ABB RobotStudio station: Mark 4.rspag

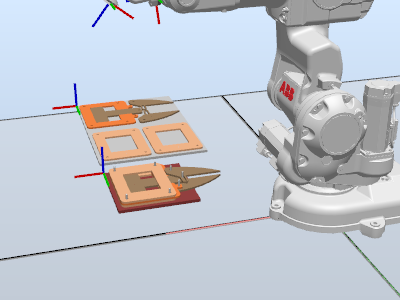
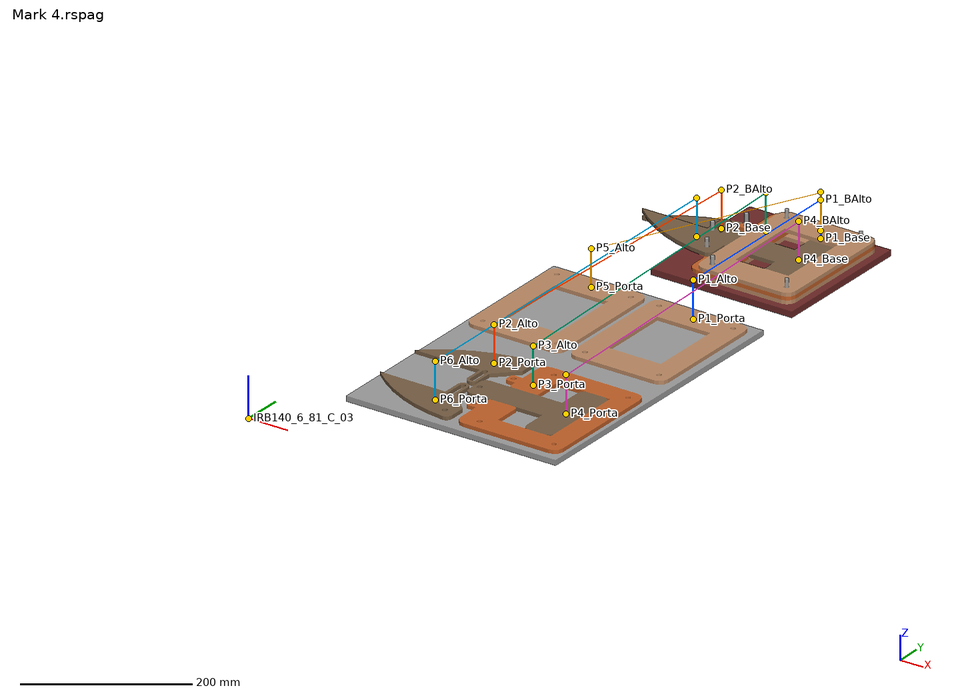
[picture v1: parts stored in the station drawn from their meshes, with robot base, taught points and paths (robot models come from the ABB library and are not in the file)]
--- station ---
Station Mark 4 (saved by RobotStudio 22.2.9947.0)
Controller Mark4_PF
  mechanical unit ROB_1: IRB140_6_81_C_03, 6 joints, base frame (0, 0, 0) mm
Layout (positions relative to the parent item):
  - IRB140_6_81_C_03 [mechanism, from Robots\IRB140_6_81_C_G_03.rslib] at (0, 0, 0) mm; joint values [0, 0, 0, 0, 0.1225, 0] (rad or m)
  - Base [part] at (585, 215, 277) mm, rotated rx 0 ry 0 rz 180 deg, size 282.5 x 200 x 35 mm
  - Portapiezas [part] at (550, -150, 277) mm, rotated rx 0 ry 0 rz 180 deg, size 297 x 420 x 12 mm
  - Tool_AJDJ [mechanism] at (514.51, 0, 704.06) mm, rotated rx 180 ry 82.98 rz 180 deg
      TCP Tool_AJDJ at (-6, 0, 116) mm, rotated rx 0 ry 45 rz 0 deg
      links: Herramienta
Attachment: Tool_AJDJ is attached to IRB140_6_81_C_03 / Link6

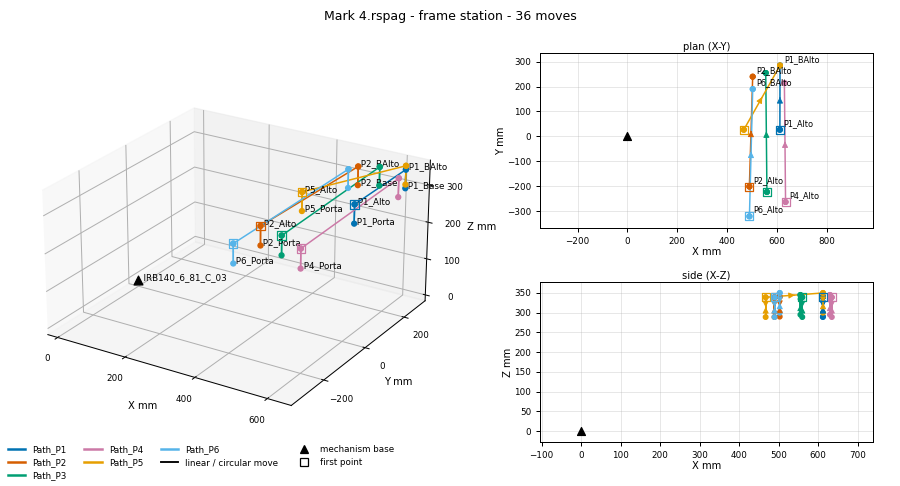
[picture p0: tool path of Mark 4.rspag in frame station, 36 of 39 moves have a stored position in this frame; points joined in program order, loops and branches not executed]
--- Backups/Mark4_PF/RAPID/TASK1/PROGMOD/CalibData.mod ---
MODULE CalibData
    PERS tooldata Tool_AJDJ:=[TRUE,[[-6,0,116],[0.923879533,0,0.382683432,0]],[0.15,[0,0,1],[1,0,0,0],0,0,0]];
    TASK PERS wobjdata Portapiezas:=[FALSE,TRUE,"",[[688.989,-362.504,284],[1,0,0,0]],[[0,0,0],[1,0,0,0]]];
    TASK PERS wobjdata BaseG:=[FALSE,TRUE,"",[[689.264,115.06,285],[1,0,0,0]],[[0,0,0],[1,0,0,0]]];
ENDMODULE

--- Backups/Mark4_PF/RAPID/TASK1/PROGMOD/Module1.mod ---
MODULE Module1
    CONST jointtarget HomeHerramienta:=[[0,0,0,0,45,0],[9E+09,9E+09,9E+09,9E+09,9E+09,9E+09]];
    CONST robtarget P1_Alto:=[[-77.3,389.019,55],[0,0,1,0],[0,-1,0,0],[9E+09,9E+09,9E+09,9E+09,9E+09,9E+09]];
    CONST robtarget P1_Porta:=[[-77.3,389.019,5],[0,0,1,0],[0,-2,1,0],[9E+09,9E+09,9E+09,9E+09,9E+09,9E+09]];
    CONST robtarget P1_BAlto:=[[-77.1,169.1,55],[0,0,1,0],[0,-1,0,0],[9E+09,9E+09,9E+09,9E+09,9E+09,9E+09]];
    CONST robtarget P1_Base:=[[-77.1,169.1,5],[0,0,1,0],[0,-1,0,0],[9E+09,9E+09,9E+09,9E+09,9E+09,9E+09]];
    CONST jointtarget HomeLaboratorio:=[[0,0,0,0,0,0],[9E+09,9E+09,9E+09,9E+09,9E+09,9E+09]];
    CONST robtarget P2_Alto:=[[-199.7,161,55],[0,0,1,0],[-1,0,-1,0],[9E+09,9E+09,9E+09,9E+09,9E+09,9E+09]];
    CONST robtarget P2_Porta:=[[-199.7,161,5],[0,0,1,0],[-1,1,-2,0],[9E+09,9E+09,9E+09,9E+09,9E+09,9E+09]];
    CONST robtarget P2_BAlto:=[[-186.7,124.4,55],[0,0,1,0],[0,-1,0,0],[9E+09,9E+09,9E+09,9E+09,9E+09,9E+09]];
    CONST robtarget P2_Base:=[[-186.7,124.4,5],[0,0,1,0],[0,-1,1,0],[9E+09,9E+09,9E+09,9E+09,9E+09,9E+09]];
    CONST robtarget P3_Alto:=[[-129.3,139.3,55],[0,0,1,0],[-1,0,-1,0],[9E+09,9E+09,9E+09,9E+09,9E+09,9E+09]];
    CONST robtarget P3_Porta:=[[-129.3,139.3,5],[0,0,1,0],[-1,0,-2,0],[9E+09,9E+09,9E+09,9E+09,9E+09,9E+09]];
    CONST robtarget P3_BAlto:=[[-134.3,139.3,60],[0,0,1,0],[0,-1,0,0],[9E+09,9E+09,9E+09,9E+09,9E+09,9E+09]];
    CONST robtarget P3_Base:=[[-134.3,139.3,10],[0,0,1,0],[0,-1,1,0],[9E+09,9E+09,9E+09,9E+09,9E+09,9E+09]];
    CONST robtarget P4_Alto:=[[-54.5,99.1,55],[0,0,1,0],[-1,0,-1,0],[9E+09,9E+09,9E+09,9E+09,9E+09,9E+09]];
    CONST robtarget P4_Porta:=[[-54.5,99.1,5],[0,0,1,0],[-1,0,-1,0],[9E+09,9E+09,9E+09,9E+09,9E+09,9E+09]];
    CONST robtarget P4_BAlto:=[[-59.5,99.1,60],[0,0,1,0],[0,-1,0,0],[9E+09,9E+09,9E+09,9E+09,9E+09,9E+09]];
    CONST robtarget P4_Base:=[[-59.5,99.1,10],[0,0,1,0],[0,-1,0,0],[9E+09,9E+09,9E+09,9E+09,9E+09,9E+09]];
    CONST robtarget P5_Alto:=[[-222,389.1,55],[0,0,1,0],[0,-1,0,0],[9E+09,9E+09,9E+09,9E+09,9E+09,9E+09]];
    CONST robtarget P5_Porta:=[[-222,389.1,5],[0,0,1,0],[0,-2,1,0],[9E+09,9E+09,9E+09,9E+09,9E+09,9E+09]];
    CONST robtarget P5_BAlto:=[[-77.1,169.1,65],[0,0,1,0],[0,-1,0,0],[9E+09,9E+09,9E+09,9E+09,9E+09,9E+09]];
    CONST robtarget P5_Base:=[[-77.1,169.1,15],[0,0,1,0],[0,-1,0,0],[9E+09,9E+09,9E+09,9E+09,9E+09,9E+09]];
    CONST robtarget P6_Alto:=[[-199.5,41.5,55],[0,0,1,0],[-1,0,-2,0],[9E+09,9E+09,9E+09,9E+09,9E+09,9E+09]];
    CONST robtarget P6_Porta:=[[-199.5,41.5,5],[0,0,1,0],[-1,0,-2,0],[9E+09,9E+09,9E+09,9E+09,9E+09,9E+09]];
    CONST robtarget P6_BAlto:=[[-186.6,74.6,65],[0,0,1,0],[0,-1,0,0],[9E+09,9E+09,9E+09,9E+09,9E+09,9E+09]];
    CONST robtarget P6_Base:=[[-186.6,74.6,15],[0,0,1,0],[0,-1,1,0],[9E+09,9E+09,9E+09,9E+09,9E+09,9E+09]];
    PROC ToHome()
        MoveAbsJ HomeLaboratorio,v150,z10,Tool_AJDJ\WObj:=BaseG;
    ENDPROC
    PROC Path_P1()
        MoveAbsJ HomeHerramienta,v150,z10,Tool_AJDJ\WObj:=BaseG;
        MoveL P1_Alto,v150,z10,Tool_AJDJ\WObj:=Portapiezas;
        MoveL P1_Porta,v50,z10,Tool_AJDJ\WObj:=Portapiezas;
        WaitDI DI_01,1;
        SetDO DO_01,1;
        WaitTime 0.05;
        SetDO DO_01,0;
        MoveL P1_Alto,v50,z10,Tool_AJDJ\WObj:=Portapiezas;
        MoveL P1_BAlto,v150,z10,Tool_AJDJ\WObj:=BaseG;
        MoveL P1_Base,v50,z10,Tool_AJDJ\WObj:=BaseG;
        WaitDI DI_01,1;
        SetDO DO_02,1;
        WaitTime 0.05;
        SetDO DO_02,0;
        MoveL P1_BAlto,v50,z10,Tool_AJDJ\WObj:=BaseG;
    ENDPROC
    PROC Path_P2()
        MoveL P2_Alto,v150,z10,Tool_AJDJ\WObj:=Portapiezas;
        MoveL P2_Porta,v50,z10,Tool_AJDJ\WObj:=Portapiezas;
        WaitDI DI_01,1;
        SetDO DO_01,1;
        WaitTime 0.05;
        SetDO DO_01,0;
        MoveL P2_Alto,v50,z10,Tool_AJDJ\WObj:=Portapiezas;
        MoveL P2_BAlto,v150,z10,Tool_AJDJ\WObj:=BaseG;
        MoveL P2_Base,v50,z10,Tool_AJDJ\WObj:=BaseG;
        WaitDI DI_01,1;
        SetDO DO_02,1;
        WaitTime 0.05;
        SetDO DO_02,0;
        MoveL P2_BAlto,v50,z10,Tool_AJDJ\WObj:=BaseG;
    ENDPROC
    PROC Path_P3()
        MoveL P3_Alto,v150,z10,Tool_AJDJ\WObj:=Portapiezas;
        MoveL P3_Porta,v50,z10,Tool_AJDJ\WObj:=Portapiezas;
        WaitDI DI_01,1;
        SetDO DO_01,1;
        WaitTime 0.05;
        SetDO DO_01,0;
        MoveL P3_Alto,v50,z10,Tool_AJDJ\WObj:=Portapiezas;
        MoveL P3_BAlto,v150,z10,Tool_AJDJ\WObj:=BaseG;
        MoveL P3_Base,v50,z10,Tool_AJDJ\WObj:=BaseG;
        WaitDI DI_01,1;
        SetDO DO_02,1;
        WaitTime 0.05;
        SetDO DO_02,0;
        MoveL P3_BAlto,v50,z10,Tool_AJDJ\WObj:=BaseG;
    ENDPROC
    PROC Path_P4()
        MoveL P4_Alto,v150,z10,Tool_AJDJ\WObj:=Portapiezas;
        MoveL P4_Porta,v50,z10,Tool_AJDJ\WObj:=Portapiezas;
        WaitDI DI_01,1;
        SetDO DO_01,1;
        WaitTime 0.05;
        SetDO DO_01,0;
        MoveL P4_Alto,v50,z10,Tool_AJDJ\WObj:=Portapiezas;
        MoveL P4_BAlto,v150,z10,Tool_AJDJ\WObj:=BaseG;
        MoveL P4_Base,v50,z10,Tool_AJDJ\WObj:=BaseG;
        WaitDI DI_01,1;
        SetDO DO_02,1;
        WaitTime 0.05;
        SetDO DO_02,0;
        MoveL P4_BAlto,v50,z10,Tool_AJDJ\WObj:=BaseG;
    ENDPROC
    PROC Path_P5()
        MoveL P5_Alto,v150,z10,Tool_AJDJ\WObj:=Portapiezas;
        MoveL P5_Porta,v50,z10,Tool_AJDJ\WObj:=Portapiezas;
        WaitDI DI_01,1;
        SetDO DO_01,1;
        WaitTime 0.05;
        SetDO DO_01,0;
        MoveL P5_Alto,v50,z10,Tool_AJDJ\WObj:=Portapiezas;
        MoveL P5_BAlto,v150,z10,Tool_AJDJ\WObj:=BaseG;
        MoveL P5_Base,v50,z10,Tool_AJDJ\WObj:=BaseG;
        WaitDI DI_01,1;
        SetDO DO_02,1;
        WaitTime 0.05;
        SetDO DO_02,0;
        MoveL P5_BAlto,v50,z10,Tool_AJDJ\WObj:=BaseG;
    ENDPROC
    PROC Path_P6()
        MoveL P6_Alto,v150,z10,Tool_AJDJ\WObj:=Portapiezas;
        MoveL P6_Porta,v50,z10,Tool_AJDJ\WObj:=Portapiezas;
        WaitDI DI_01,1;
        SetDO DO_01,1;
        WaitTime 0.05;
        SetDO DO_01,0;
        MoveL P6_Alto,v50,z10,Tool_AJDJ\WObj:=Portapiezas;
        MoveL P6_BAlto,v150,z10,Tool_AJDJ\WObj:=BaseG;
        MoveL P6_Base,v50,z10,Tool_AJDJ\WObj:=BaseG;
        WaitDI DI_01,1;
        SetDO DO_02,1;
        WaitTime 0.05;
        SetDO DO_02,0;
        MoveL P6_BAlto,v50,z10,Tool_AJDJ\WObj:=BaseG;
        MoveAbsJ HomeHerramienta,v150,z10,Tool_AJDJ\WObj:=BaseG;
    ENDPROC
    PROC main()
        SpyStart "HOME:/spy.log";
        SetDO DO_03,0;
        WaitDI DI_01,1;
        ToHome;
        WaitDI DI_01,1;
        Path_P1;
        Path_P2;
        Path_P3;
        Path_P4;
        Path_P5;
        Path_P6;
        ToHome;
        SetDO DO_03,1;
        SpyStop;
        Break;
    ENDPROC
ENDMODULE

--- Backups/Mark4_PF/SYSPAR/EIO.cfg ---
EIO:CFG_1.0:6:1::
#
EIO_SIGNAL:

      -Name "DI_01" -SignalType "DI"

      -Name "DO_01" -SignalType "DO"

      -Name "DO_02" -SignalType "DO"

      -Name "DO_03" -SignalType "DO"
